FUNCTION_BLOCK FB_DevicesV2 

VAR

END_VAR

//INITIEREN

//Kleppen

//Object dat het waterpeil berekend


//Object wat een gewenst debiet kan simuleren


//Object dat de kleppen regelt

END_FUNCTION_BLOCK

(* stored: Version 1.1.0.1, ProductVersion 3.1.4024.12
   POU FB_DevicesV2: Id {274ae7ad-92b9-47e2-b334-e236e1093c9f}, SpecialFunc None *)
